GLOBALCONSTANTS TCPool (* Global constants *)
  (* Standard: 61499-1 *)
  (* Version 1.0, 2024-02-25, franz *)
  VAR_GLOBAL CONSTANT
    DE_NUM_DEVICE : UINT := 0;
    DE_NUM_CONN : UINT := 10;
    DE_NUM_SECTION_001 : UINT := 11;
    DE_NUM_SECTION_002 : UINT := 12;
    DE_NUM_SECTION_003 : UINT := 13;
    DE_NUM_SECTION_004 : UINT := 14;
    DE_NUM_SECTION_005 : UINT := 15;
    DE_NUM_SECTION_006 : UINT := 16;
    DE_NUM_SECTION_007 : UINT := 17;
    DE_NUM_SECTION_008 : UINT := 18;
    DE_NUM_SECTION_009 : UINT := 19;
    DE_NUM_SECTION_010 : UINT := 20;
    DE_NUM_SECTION_011 : UINT := 21;
    DE_NUM_SECTION_012 : UINT := 22;
    DE_NUM_SECTION_013 : UINT := 23;
    DE_NUM_SECTION_014 : UINT := 24;
    DE_NUM_SECTION_015 : UINT := 25;
    DE_NUM_SECTION_016 : UINT := 26;
    OBJID_DET_DEVICE : UINT := 100;
    OBJID_DET_CONN : UINT := 101;
    OBJID_DET_SECTION_001 : UINT := 102;
    OBJID_DET_SECTION_002 : UINT := 103;
    OBJID_DET_SECTION_003 : UINT := 104;
    OBJID_DET_SECTION_004 : UINT := 105;
    OBJID_DET_SECTION_005 : UINT := 106;
    OBJID_DET_SECTION_006 : UINT := 107;
    OBJID_DET_SECTION_007 : UINT := 108;
    OBJID_DET_SECTION_008 : UINT := 109;
    OBJID_DET_SECTION_009 : UINT := 110;
    OBJID_DET_SECTION_010 : UINT := 111;
    OBJID_DET_SECTION_011 : UINT := 112;
    OBJID_DET_SECTION_012 : UINT := 113;
    OBJID_DET_SECTION_013 : UINT := 114;
    OBJID_DET_SECTION_014 : UINT := 115;
    OBJID_DET_SECTION_015 : UINT := 116;
    OBJID_DET_SECTION_016 : UINT := 117;
    OBJID_DPD_ACTUAL_WORK_STATE : UINT := 118;
    OBJID_DPD_MAXIMUM_WORKING_WIDTH : UINT := 119;
    OBJID_DPD_ACTUAL_WORKING_WIDTH : UINT := 120;
    OBJID_DPD_ACTUAL_WORKING_WIDTH_SECTION : UINT := 121;
    OBJID_DPD_OFFSET_X_BOOM : UINT := 122;
    OBJID_DPD_OFFSET_Y_BOOM : UINT := 123;
    OBJID_DPD_PRESCRIPTION_CONTROL_STATE : UINT := 124;
    OBJID_DPD_SECTION_CONTROL_STATE : UINT := 125;
    OBJID_DPD_ACTUAL_CONDENSED_WORK_STATE_1_16 : UINT := 126;
    OBJID_DPD_SETPOINT_CONDENSED_WORK_STATE_1_16 : UINT := 127;
    OBJID_DPD_OFFSET_X_CONNECTOR : UINT := 128;
    OBJID_DPD_OFFSET_Y_CONNECTOR : UINT := 129;
    OBJID_DPD_CONNECTOR_TYPE : UINT := 130;
    OBJID_DPD_OFFSET_X_SECTION : UINT := 131;
    OBJID_DPD_OFFSET_Y_SECTION_001 : UINT := 132;
    OBJID_DPD_OFFSET_Y_SECTION_002 : UINT := 133;
    OBJID_DPD_OFFSET_Y_SECTION_003 : UINT := 134;
    OBJID_DPD_OFFSET_Y_SECTION_004 : UINT := 135;
    OBJID_DPD_OFFSET_Y_SECTION_005 : UINT := 136;
    OBJID_DPD_OFFSET_Y_SECTION_006 : UINT := 137;
    OBJID_DPD_OFFSET_Y_SECTION_007 : UINT := 138;
    OBJID_DPD_OFFSET_Y_SECTION_008 : UINT := 139;
    OBJID_DPD_OFFSET_Y_SECTION_009 : UINT := 140;
    OBJID_DPD_OFFSET_Y_SECTION_010 : UINT := 141;
    OBJID_DPD_OFFSET_Y_SECTION_011 : UINT := 142;
    OBJID_DPD_OFFSET_Y_SECTION_012 : UINT := 143;
    OBJID_DPD_OFFSET_Y_SECTION_013 : UINT := 144;
    OBJID_DPD_OFFSET_Y_SECTION_014 : UINT := 145;
    OBJID_DPD_OFFSET_Y_SECTION_015 : UINT := 146;
    OBJID_DPD_OFFSET_Y_SECTION_016 : UINT := 147;
    OBJID_DPD_SETPOINT : UINT := 148;
    OBJID_DPD_ACTUAL : UINT := 149;
    OBJID_DPD_ACTUAL_CULTURAL_PRACTICE : UINT := 150;
    OBJID_DPD_HAUL_COUNTER : UINT := 151; (* 464 - Haul Counter *)
    OBJID_DPD_LIFETIME_HAUL_COUNTER : UINT := 152; (* 465 - Lifetime Haul Counter *)
    OBJID_DPD_TOTAL_AREA : UINT := 153; (* DDI 116 *)
    OBJID_DPD_TOTAL_DISTANCE : UINT := 154; (* DDI 597 *)
    OBJID_DPD_EFFECTIVE_TOTAL_DISTANCE : UINT := 155; (* DDI 117 *)
    OBJID_DPD_TOTAL_DISTANCE_FIELD : UINT := 156; (* DDI 599 *)
    OBJID_DPD_INEFFECTIVE_TOTAL_DISTANCE : UINT := 157; (* DDI 118 *)
    OBJID_DPD_TOTAL_DISTANCE_STREET : UINT := 158; (* DDI 601 *)
    OBJID_DPD_EFFECTIVE_TOTAL_TIME : UINT := 159; (* DDI 119 *)
    OBJID_DPD_INEFFECTIVE_TOTAL_TIME : UINT := 160; (* DDI 120 *)
    OBJID_DPD_LIFETIME_TOTAL_AREA : UINT := 161; (* DDI 271 *)
    OBJID_DPD_LIFETIME_TOTAL_DISTANCE : UINT := 162; (* DDI 598 *)
    OBJID_DPD_LIFETIME_EFFECTIVE_TOTAL_DISTANCE : UINT := 163; (* DDI 272 *)
    OBJID_DPD_LIFETIME_TOTAL_DISTANCE_FIELD : UINT := 164; (* DDI 600 *)
    OBJID_DPD_LIFETIME_INEFFECTIVE_TOTAL_DISTANCE : UINT := 165; (* DDI 273 *)
    OBJID_DPD_LIFETIME_TOTAL_DISTANCE_STREET : UINT := 166; (* DDI 602 *)
    OBJID_DPD_LIFETIME_EFFECTIVE_TOTAL_TIME : UINT := 167; (* DDI 274 *)
    OBJID_DPD_LIFETIME_INEFFECTIVE_TOTAL_TIME : UINT := 168; (* DDI 275 *)
    OBJID_DVP_ACTUAL_WORK_STATE : UINT := 169;
    OBJID_DVP_UNIT_M : UINT := 170;
    OBJID_DVP_UNIT_HOUR : UINT := 171;
    OBJID_DVP_UNIT_SEC : UINT := 172;
    OBJID_DVP_UNIT_HA : UINT := 173;
    OBJID_DVP_UNIT_HAUL_COUNTER : UINT := 174;
    OBJID_DPD_DEFAULT_DDI : UINT := 59999;
    OBJID_DVP_NO_UNIT : UINT := 16#FFFF;
  END_VAR
END_GLOBALCONSTANTS
